{attribute 'GeneratedUsingTerminal: EL3692-0000-0017'}
{attribute addProperty BoxType "EL3692-0000-0017"}
{attribute addProperty Id "StatusAT %I*Status_439F40C310ValueAT %I*DINT4"}
{attribute addProperty CRC "2647483735"}
{attribute addProperty Size "14"}
TYPE SAI_Inputs_Channel_9DCD6557 :
STRUCT
	{attribute addProperty Name "Status"}
	Status AT %I* : Status_439F40C3;
	{attribute addProperty Name "Value"}
	Value AT %I* : DINT;
END_STRUCT
END_TYPE

(* stored: Version 1.2.0.0, ProductVersion 3.1.4024.9
   DUT SAI_Inputs_Channel_9DCD6557: Id {5cbf7b7d-4ffe-4132-8d99-bd10459f6a40} *)
